FUNCTION_BLOCK PASS_COLOUR (* Basic Function Block Type *)
  (* Standard: 61499-2 *)
  (* Version 0.3, 2009-09-15, JHC, Holobloc Inc, Changed transition priorities. *)
  (* Version 0.2, 2003-12-04, JHC, Rockwell Automation, Renamed for better indexing. *)
  (* Version 0.1, 2002-11-05, JHC, Rockwell Automation, Corrected missing ST element in Algorithm REQ. *)
  (* Version 0.0, 2000-05-30, JHC, Rockwell Automation *)
  (* Compiler header: package fb.rt.template; *)
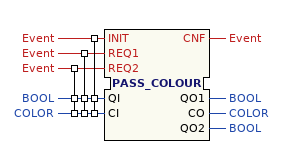
  EVENT_INPUT
    INIT WITH QI, CI; (* Initialization Request *)
    REQ1 WITH QI, CI; (* Normal Execution Request *)
    REQ2 WITH QI, CI;
  END_EVENT
  EVENT_OUTPUT
    CNF;
  END_EVENT
  VAR_INPUT
    QI : BOOL; (* Input event qualifier *)
    CI : COLOR;
  END_VAR
  VAR_OUTPUT
    QO1 : BOOL; (* Output event qualifier *)
    CO : COLOR;
    QO2 : BOOL;
  END_VAR
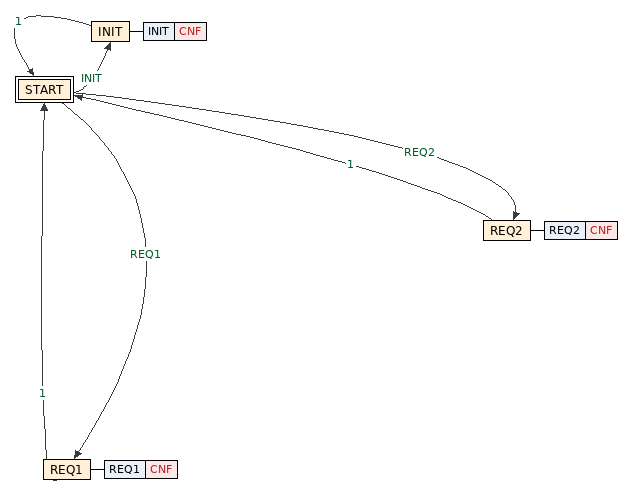
  EC_STATES
    START; (* Initial State *)
    INIT : INIT -> CNF; (* Initialization *)
    REQ1 : REQ1 -> CNF; (* Normal execution *)
    REQ2 : REQ2 -> CNF;
  END_STATES
  EC_TRANSITIONS
    INIT TO START := 1;
    START TO REQ1 := REQ1;
    START TO INIT := INIT;
    REQ1 TO START := 1;
    START TO REQ2 := REQ2;
    REQ2 TO START := 1;
  END_TRANSITIONS
  ALGORITHM INIT IN Java: (* Initialization algorithm *)
QO1.value=false;
QO2.value=true;
CO.value=CI.value;
  END_ALGORITHM
  ALGORITHM REQ1 IN Java: (* Normally executed algorithm *)
QO1.value=QI.value;
QO2.value=QI.value;
CI.value=CO.value;
  END_ALGORITHM
  ALGORITHM REQ2 IN ST:
QO2:=FALSE;
QO1:=QI;
  END_ALGORITHM
END_FUNCTION_BLOCK
